{attribute addProperty BoxType "EL3311-0000-0018"}
{attribute addProperty Id "TC_InputsAT %I*TC_Inputs_FFD159D63240WcStateAT %I*WcState_F855686C1620InfoDataAT %I*InfoData_BC63D37F80100"}
{attribute addProperty CRC "3559080678"}
{attribute addProperty SizeInBites "128"}
{attribute addProperty SizeInBytes "16"}
TYPE EL3311_18CEA68E :
STRUCT
	{attribute addProperty Name "TC_Inputs"}
	TC_Inputs : TC_Inputs_FFD159D6;
	{attribute addProperty Name "WcState"}
	WcState : WcState_F855686C;
	{attribute addProperty Name "InfoData"}
	InfoData : InfoData_BC63D37F;
END_STRUCT
END_TYPE

(* stored: Version 1.2.0.0, ProductVersion 3.1.4024.9
   DUT EL3311_18CEA68E: Id {d7cdb7f0-b9da-4849-8cb9-14cae659cb1e} *)
